INTERFACE I_Domain EXTENDS Debug.I_Debug, Tags.I_Tagged

PROPERTY Flags : Flags.I_FlagList
GET
END_GET
END_PROPERTY

PROPERTY Recs : Broadcast.I_ReceiverList
GET
END_GET
END_PROPERTY

PROPERTY Signals : Broadcast.I_SignalList
GET
END_GET
END_PROPERTY

PROPERTY Smgr : States.I_StateManager
GET
END_GET
END_PROPERTY

END_INTERFACE

(* stored: Version 1.1.0.1
   Itf I_Domain: Id {83fc7eee-7760-4606-8251-3726a07db91d}
   Property Flags: Id {0d61cdfd-ef8a-441b-b785-3063266e4226}
   Get Get: Id {20ec1d7e-7c8b-4ef0-a987-d90a1bb5c12e}
   Property Recs: Id {a93da77b-5c4b-4b94-8689-c988ae5a90fe}
   Get Get: Id {009bf5c3-8701-4f7a-b3e1-aa09cf3c3339}
   Property Signals: Id {a556fd7f-828c-49b0-9a3e-cfe8bbf10ffd}
   Get Get: Id {38a4b043-5c44-4b32-8064-f02b53f04fa1}
   Property Smgr: Id {5fea3b40-e370-410d-8034-700858b6c408}
   Get Get: Id {0216a31d-0aa3-497d-b609-80d8d44d44b5} *)
